PROGRAM Q2
VAR
	tempurature : REAL := 26.5;
END_VAR

END_PROGRAM

(* stored: Version 1.1.0.1, ProductVersion 3.1.4024.12
   POU Q2: Id {697cbeb6-d739-4545-9ae0-31c7cee95e84}, SpecialFunc None *)
